PROGRAM TrafficManager
VAR
Simulator: Cars;
UpdateLights: Kims_UpdateLights;
runOnce:BOOL:=FALSE;
END_VAR

METHOD Change_TrafficFlow : BOOL
VAR_INPUT
	Intersect: POINTER to Intersection;
	NewNS_Density, NewEW_Density: TrafficDensity;
	Exit1, Exit2: Compass;
END_VAR
Intersect^.NS_Road:= NewNS_Density;
Intersect^.EW_Road:= NewEW_Density;
Intersect^.Exit1 := Exit1;
Intersect^.Exit2 := Exit2;
END_METHOD

METHOD Init : BOOL
VAR_INPUT
	//First, Second, Main, Pine :TrafficDensity;
END_VAR
//FirstAndMain.NS_Road:=TrafficDensity.Low;
//FirstAndMain.EW_Road:=TrafficDensity.Medium;
//FirstAndMain.Exit1:= North;
//FirstAndMain.Exit2:= West;
Change_TrafficFlow(ADR(FirstAndMain),TrafficDensity.Low,TrafficDensity.Medium, North, West);
Change_TrafficFlow(ADR(SecondAndMain),TrafficDensity.Medium,TrafficDensity.Medium, North, East);

Change_TrafficFlow(ADR(FirstAndPine),TrafficDensity.Low,TrafficDensity.High, South, West);
Change_TrafficFlow(ADR(SecondAndPine),TrafficDensity.Medium,TrafficDensity.High, South, East);
END_METHOD

METHOD Update
VAR_INPUT
END_VAR
UpdateLights(Intersect:=ADR(FirstAndMain));
UpdateLights(Intersect:=ADR(SecondAndMain));
//			  |						   |
//---------------<-Main Street->------------------
//		First |					Second |
//			  |						   |
//			  |  					   |
//----------------<-Pine Street->------------------
//			  |						   |
UpdateLights(Intersect:=ADR(FirstAndPine));
UpdateLights(Intersect:=ADR(SecondAndPine));


//Below this point I'm just Playing with my Hot Wheels haha//
Simulator.AddCars(ADR(FirstAndMain));
Simulator.AddCars(ADR(SecondAndMain));
Simulator.AddCars(ADR(FirstAndPine));
Simulator.AddCars(ADR(SecondAndPine));
Simulator.MoveCars(ADR(FirstAndMain), ADR(SecondAndMain), Compass.East, ADR(FirstAndPine), Compass.South);
Simulator.MoveCars(ADR(SecondAndPine), ADR(SecondAndMain), Compass.North, ADR(FirstAndPine), Compass.West);
END_METHOD

END_PROGRAM

(* stored: Version 1.1.0.1, ProductVersion 3.1.4024.11
   POU TrafficManager: Id {f9cd464c-baa3-4ab8-8ab5-576788caeb1f}, SpecialFunc None
   Method Change_TrafficFlow: Id {34aea9bc-4842-4d51-8488-552182821f60}
   Method Init: Id {4af402df-6d40-4d47-9111-d375f8a9ea95}
   Method Update: Id {8e35d2c6-934a-4647-9bfc-9e09ec83a63a} *)
